// TIA Portal V15.1 export
// export: Created 2020-06-12T07:35:53.0068359Z, ExportSetting None, DisplayName Totally Integrated Automation Portal, DisplayVersion V15.1, DisplayName TIA Portal Openness, DisplayVersion V15.1, DisplayName STEP 7 Professional, DisplayVersion V15.1, DisplayName STEP 7 Safety, DisplayVersion V15.1, DisplayName WinCC Advanced, DisplayVersion V15.1
FUNCTION "MELT_Time" : Void   // FC122, FBD
{ S7_Optimized_Access := 'TRUE' }
// stored: SetENOAutomatically False
   VAR_TEMP
      _tmp_time : Time;
      _t_mr_time : Time;
      _left_tot : Real;
      _left_mt : Real;
      _dur_tot : Real;
      _dur_mt : Real;
      tHTProgress : Real;
      tClock1 : Bool;
      tClock2 : Bool;
      tTime1 : Real;
      tTime2 : Real;
      tToRemeltWeight : Real;
      tReqVentilation : Bool;
      tMRs : Real;
      tEnCalc1 : Bool;
      tEnCalc2 : Bool;
      tMRbase : Real;
      tMRht : Real;
      tTbase : Real;
      tTht : Real;
      tTtotal : Real;
      tHTWeight : Real;
   END_VAR
BEGIN

REGION Network 1: Enable the calculations (1)
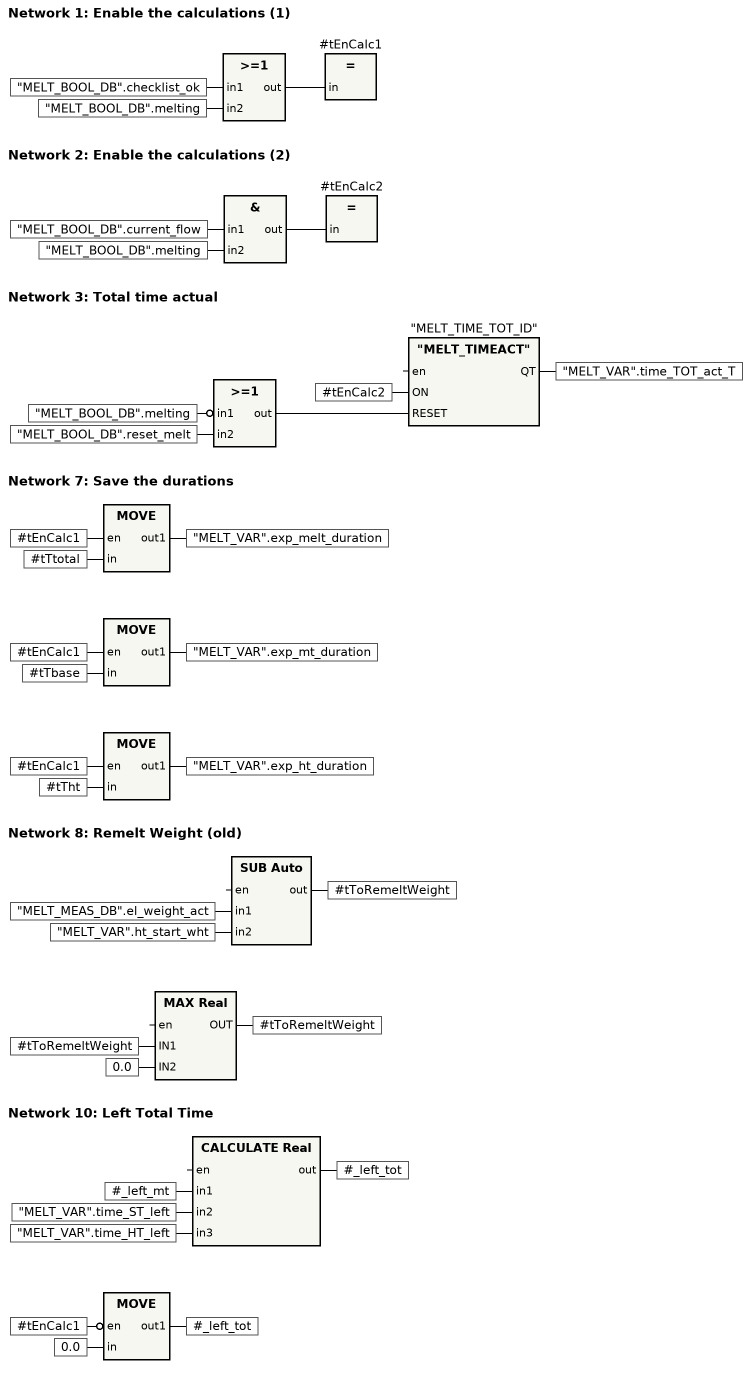
   #tEnCalc1 := "MELT_BOOL_DB".checklist_ok OR "MELT_BOOL_DB".melting;
END_REGION

REGION Network 2: Enable the calculations (2)
   #tEnCalc2 := "MELT_BOOL_DB".current_flow AND "MELT_BOOL_DB".melting;
END_REGION

REGION Network 3: Total time actual
   // VLS: delete "end_melt" from RESET time
   "MELT_TIME_TOT_ID"(ON := #tEnCalc2,   // "MELT_TIMEACT"
                      RESET := NOT "MELT_BOOL_DB".melting OR "MELT_BOOL_DB".reset_melt,
                      QT => "MELT_VAR".time_TOT_act_T);
END_REGION

REGION Network 4 (SCL): Remelt Weight (new)
   #tToRemeltWeight := "MELT_MEAS_DB".el_weight_tared;
   #tToRemeltWeight := #tToRemeltWeight - "MELT_VAR".ht_start_wht;
   IF #tToRemeltWeight < 1 THEN
       #tToRemeltWeight := 0.0;
   END_IF;
   #tHTWeight := "MELT_VAR".ht_start_wht - "MELT_VAR".ht_stop_wht;
END_REGION

REGION Network 5 (SCL): Meltrate correction for the every phase
   IF #tEnCalc1 AND "MELT_BOOL_DB".melt_main_phase THEN
       #tMRbase := "MELT_CONT_DB".mr_set * 0.5 + "MELT_CONT_DB".mr_act * 0.5;
   ELSE
       #tMRbase := "MELT_CONT_DB".mr_set;
   END_IF;
   #tMRht := #tMRbase * 0.55;
END_REGION

REGION Network 6 (SCL): Calculate the duration
   #tTbase := #tToRemeltWeight / #tMRbase * 60.0;
   #tTht := MIN(IN1 := #tHTWeight / #tMRht * 60.0, IN2 := "MELT_VAR".curve_HT_PR_tmax);
   #tTtotal := "MELT_VAR".curve_ST_P_tmax + #tTbase + #tTht;
END_REGION

REGION Network 7: Save the durations
   IF #tEnCalc1 THEN
       "MELT_VAR".exp_melt_duration := #tTtotal;
       "MELT_VAR".exp_mt_duration := #tTbase;
       "MELT_VAR".exp_ht_duration := #tTht;
   END_IF;
END_REGION

REGION Network 8: Remelt Weight (old)
   #tToRemeltWeight := "MELT_MEAS_DB".el_weight_act - "MELT_VAR".ht_start_wht;
   #tToRemeltWeight := MAX(IN1 := #tToRemeltWeight, IN2 := 0.0);
END_REGION

REGION Network 9 (SCL): Left Time during Melt Phase
   IF #tEnCalc1 THEN
       IF "MELT_CONT_DB".mr_set > 0 THEN
           #tMRs := "MELT_CONT_DB".mr_set;
       ELSE
           #tMRs := 50.0; // default value
       END_IF;
       #_left_mt := #tToRemeltWeight / #tMRs * 60.0;
   ELSE
       #_left_mt := 0.0;
   END_IF;
END_REGION

REGION Network 10: Left Total Time
   #_left_tot := #_left_mt+"MELT_VAR".time_ST_left+"MELT_VAR".time_HT_left;
   IF NOT #tEnCalc1 THEN #_left_tot := 0.0; END_IF;
END_REGION

REGION Network 11: Duration of Melt phase
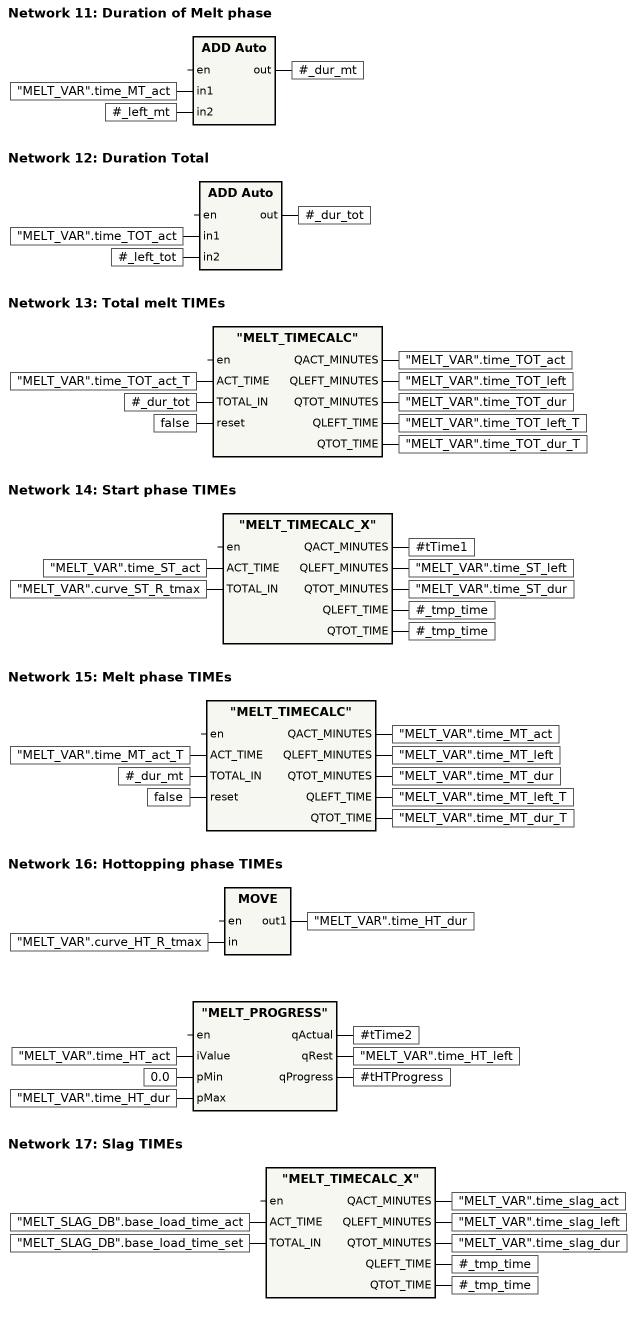
   #_dur_mt := "MELT_VAR".time_MT_act + #_left_mt;
END_REGION

REGION Network 12: Duration Total
   #_dur_tot := "MELT_VAR".time_TOT_act + #_left_tot;
END_REGION

REGION Network 13: Total melt TIMEs
   "MELT_TIMECALC"(ACT_TIME := "MELT_VAR".time_TOT_act_T,
                   TOTAL_IN := #_dur_tot,
                   reset := false,
                   QACT_MINUTES => "MELT_VAR".time_TOT_act,
                   QLEFT_MINUTES => "MELT_VAR".time_TOT_left,
                   QTOT_MINUTES => "MELT_VAR".time_TOT_dur,
                   QLEFT_TIME => "MELT_VAR".time_TOT_left_T,
                   QTOT_TIME => "MELT_VAR".time_TOT_dur_T);
END_REGION

REGION Network 14: Start phase TIMEs
   "MELT_TIMECALC_X"(ACT_TIME := "MELT_VAR".time_ST_act,
                     TOTAL_IN := "MELT_VAR".curve_ST_R_tmax,
                     QACT_MINUTES => #tTime1,
                     QLEFT_MINUTES => "MELT_VAR".time_ST_left,
                     QTOT_MINUTES => "MELT_VAR".time_ST_dur,
                     QLEFT_TIME => #_tmp_time,
                     QTOT_TIME => #_tmp_time);
END_REGION

REGION Network 15: Melt phase TIMEs
   "MELT_TIMECALC"(ACT_TIME := "MELT_VAR".time_MT_act_T,
                   TOTAL_IN := #_dur_mt,
                   reset := false,
                   QACT_MINUTES => "MELT_VAR".time_MT_act,
                   QLEFT_MINUTES => "MELT_VAR".time_MT_left,
                   QTOT_MINUTES => "MELT_VAR".time_MT_dur,
                   QLEFT_TIME => "MELT_VAR".time_MT_left_T,
                   QTOT_TIME => "MELT_VAR".time_MT_dur_T);
END_REGION

REGION Network 16: Hottopping phase TIMEs
   // "MELT_VAR_DB".time_HT_dur
   "MELT_VAR".time_HT_dur := "MELT_VAR".curve_HT_R_tmax;
   "MELT_PROGRESS"(iValue := "MELT_VAR".time_HT_act,
                   pMin := 0.0,
                   pMax := "MELT_VAR".time_HT_dur,
                   qActual => #tTime2,
                   qRest => "MELT_VAR".time_HT_left,
                   qProgress => #tHTProgress);
END_REGION

REGION Network 17: Slag TIMEs
   "MELT_TIMECALC_X"(ACT_TIME := "MELT_SLAG_DB".base_load_time_act,
                     TOTAL_IN := "MELT_SLAG_DB".base_load_time_set,
                     QACT_MINUTES => "MELT_VAR".time_slag_act,
                     QLEFT_MINUTES => "MELT_VAR".time_slag_left,
                     QTOT_MINUTES => "MELT_VAR".time_slag_dur,
                     QLEFT_TIME => #_tmp_time,
                     QTOT_TIME => #_tmp_time);
END_REGION

REGION Network 18: Time in Meltphase/HT-phase
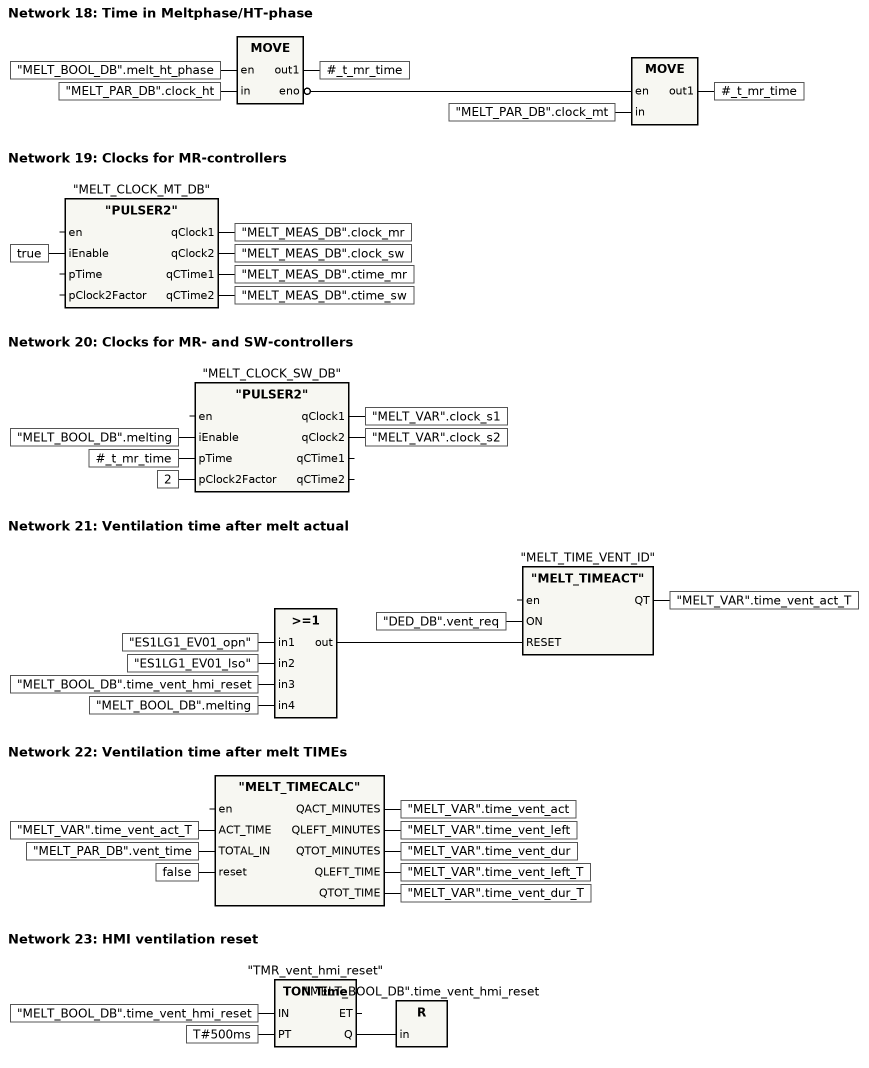
   // ENO of a box is taken as its EN; it also drops when the box reports an error
   IF "MELT_BOOL_DB".melt_ht_phase THEN #_t_mr_time := "MELT_PAR_DB".clock_ht; END_IF;
   IF NOT "MELT_BOOL_DB".melt_ht_phase THEN #_t_mr_time := "MELT_PAR_DB".clock_mt; END_IF;
END_REGION

REGION Network 19: Clocks for MR-controllers
   // TODO: link a variable {#_t_mr_time}
   // 
   // The SW-controller can work with shorter cycle time than MR-controller.
   // And the process parameters P and R depend from each other. To avoid a disturbance from a transfer procees we will use next method:
   // * MR cycle time = SW cycle time * Factor[Int >= 1]
   // * MR clock pulses has a phase (shift) relative to the SW clock pulses
   "MELT_CLOCK_MT_DB"(iEnable := true,   // "PULSER2"
                      qClock1 => "MELT_MEAS_DB".clock_mr,
                      qClock2 => "MELT_MEAS_DB".clock_sw,
                      qCTime1 => "MELT_MEAS_DB".ctime_mr,
                      qCTime2 => "MELT_MEAS_DB".ctime_sw);
END_REGION

REGION Network 20: Clocks for MR- and SW-controllers
   // TODO: link a variable {#_t_mr_time}
   // 
   // The SW-controller can work with shorter cycle time than MR-controller.
   // And the process parameters P and R depend from each other. To avoid a disturbance from a transfer procees we will use next method:
   // * MR cycle time = SW cycle time * Factor[Int >= 1]
   // * MR clock pulses has a phase (shift) relative to the SW clock pulses
   "MELT_CLOCK_SW_DB"(iEnable := "MELT_BOOL_DB".melting,   // "PULSER2"
                      pTime := #_t_mr_time,
                      pClock2Factor := 2,
                      qClock1 => "MELT_VAR".clock_s1,
                      qClock2 => "MELT_VAR".clock_s2);
END_REGION

REGION Network 21: Ventilation time after melt actual
   // "ES1LD1_EV03_opn"
   // "ES1LE3_EV06_opn"
   "MELT_TIME_VENT_ID"(ON := "DED_DB".vent_req,   // "MELT_TIMEACT"
                       RESET := "ES1LG1_EV01_opn" OR "ES1LG1_EV01_lso" OR "MELT_BOOL_DB".time_vent_hmi_reset OR "MELT_BOOL_DB".melting,
                       QT => "MELT_VAR".time_vent_act_T);
END_REGION

REGION Network 22: Ventilation time after melt TIMEs
   "MELT_TIMECALC"(ACT_TIME := "MELT_VAR".time_vent_act_T,
                   TOTAL_IN := "MELT_PAR_DB".vent_time,
                   reset := false,
                   QACT_MINUTES => "MELT_VAR".time_vent_act,
                   QLEFT_MINUTES => "MELT_VAR".time_vent_left,
                   QTOT_MINUTES => "MELT_VAR".time_vent_dur,
                   QLEFT_TIME => "MELT_VAR".time_vent_left_T,
                   QTOT_TIME => "MELT_VAR".time_vent_dur_T);
END_REGION

REGION Network 23: HMI ventilation reset
   "TMR_vent_hmi_reset".TON(IN := "MELT_BOOL_DB".time_vent_hmi_reset, PT := T#500ms);
   IF "TMR_vent_hmi_reset".Q THEN "MELT_BOOL_DB".time_vent_hmi_reset := FALSE; END_IF;
END_REGION
END_FUNCTION
